// TIA Portal project "PLCSIM15-sort-height-basic_V17" (V17)
// Vorlageprojekt für das Buch mit Zielsystem S7-1200

(* hardware
DEVICE "S7-1200-Station_1"  S7-1200 Station
   slot 0: "Baugruppenträger_0"  Rack  V1.0
   slot 1: "PLC_1"  CPU 1211C DC/DC/DC  6ES7 211-1AE40-0XB0  V4.1
*)

// ===== PLC "PLC_1"  CPU 1211C DC/DC/DC =====

VAR_GLOBAL   // PLC tag table "Standard-Variablentabelle"
   "Tag_1" AT %A0.0 : Bool;
   "Tag_2" AT %E0.0 : Bool;
   "Tag_3" AT %E0.1 : Bool;
   "Warning Light" AT %Q1.2 : Bool;
END_VAR

VAR_GLOBAL   // PLC tag table "Tag table_1"
   "I_High_sensor" AT %I0.0 : Bool;
   "I_Low_sensor" AT %I0.1 : Bool;
   "I_Pallet_sensor" AT %I0.2 : Bool;
   "I_Loaded" AT %I0.3 : Bool;
   "I_At_left_entry" AT %I0.4 : Bool;
   "I_At_left_exit" AT %I0.5 : Bool;
   "I_At_right_entry" AT %I0.6 : Bool;
   "I_At_right_exit" AT %I0.7 : Bool;
   "O_Conveyor_entry" AT %Q0.0 : Bool;
   "O_Load" AT %Q0.1 : Bool;
   "O_Unload" AT %Q0.2 : Bool;
   "O_Transf_left" AT %Q0.3 : Bool;
   "O_Tranf_right" AT %Q0.4 : Bool;
   "O_Conveyor_left" AT %Q0.5 : Bool;
   "Loading" AT %M0.0 : Bool;
   "LoaderBusy" AT %M0.1 : Bool;
   "TransferingRight" AT %M0.2 : Bool;
   "TransferingLeft" AT %M0.3 : Bool;
   "HighBox" AT %M0.4 : Bool;
   "I_Start" AT %I1.0 : Bool;
   "I_Reset" AT %I1.1 : Bool;
   "I_Stop" AT %I1.2 : Bool;
   "I_Emergency" AT %I1.3 : Bool;
   "I_Auto" AT %I1.4 : Bool;
   "I_Factory_Running" AT %I1.5 : Bool;
   "O_Conveyor_right" AT %Q0.6 : Bool;
   "O_Start_light" AT %Q0.7 : Bool;
   "O_Reset_light" AT %Q1.0 : Bool;
   "O_Stop_light" AT %Q1.1 : Bool;
   "P_High_Sensor" AT %M1.0 : Bool;
   "P_Loading" AT %M1.1 : Bool;
   "P_At_left_entry" AT %M1.4 : Bool;
   "P_At_left_exit" AT %M1.5 : Bool;
   "P_At_right_entry" AT %M1.6 : Bool;
   "P_At_right_exit" AT %M1.7 : Bool;
   "P_Factory_Running" AT %M2.5 : Bool;
   "FactoryRestarting" AT %M0.5 : Bool;
END_VAR

// folder: System blocks/Program resources

DATA_BLOCK "RightCounter"   // DB1
{ S7_Optimized_Access := 'TRUE' }
AUTHOR : Simatic
FAMILY : IEC
NAME : CNTR
VERSION : 1.0
// stored: InstanceOfName IEC_COUNTER
"IEC_COUNTER"
BEGIN
END_DATA_BLOCK

DATA_BLOCK "LeftCounter"   // DB2
{ S7_Optimized_Access := 'TRUE' }
AUTHOR : Simatic
FAMILY : IEC
NAME : CNTR
VERSION : 1.0
// stored: InstanceOfName IEC_COUNTER
"IEC_COUNTER"
BEGIN
END_DATA_BLOCK

// folder: (top level)

FUNCTION "MHJ-PLC-Lab-Function-S71200" : Void   // FC9000, SCL
{ S7_Optimized_Access := 'TRUE' }
VERSION : 0.1
   VAR_TEMP
      rdTimeReturn : Int;
      outputTime : DTL;
      SyncVal : Byte;
      forVal : Int;
      forVal_2 : Int;
      Value : Byte;
   END_VAR
   VAR CONSTANT
      CompVal : Byte := 16#34;
      Value_01 : Byte := 16#11;
      Value_01_DW : DWord := 16#A165_D992;
      Value_02_DW : DWord := 16#58BE_4401;
   END_VAR
BEGIN

   #Value:=PEEK(area := 16#82,
        dbNumber := 0,
        byteOffset := 511);
   #Value := #Value + 1;

   POKE(area := 16#82,
        dbNumber := 0,
        byteOffset := 511,
        value := #Value);

   POKE(area:=16#81,
        dbNumber:=0,
        byteOffset:=1016,
        value:=#Value_01_DW);
   POKE(area := 16#81,
        dbNumber := 0,
        byteOffset := 1020,
        value := #Value_02_DW);

   POKE(area := 16#81,
        dbNumber := 0,
        byteOffset := 511,
        value := B#16#00);

   FOR #forVal := 0 TO 120 DO
       FOR #forVal_2:=0 TO 10 DO
           #rdTimeReturn:=RD_SYS_T(#outputTime);
           #rdTimeReturn := WR_SYS_T(#outputTime);
           #rdTimeReturn := RD_SYS_T(#outputTime);
           #rdTimeReturn := WR_SYS_T(#outputTime);
       END_FOR;
       #SyncVal:= PEEK(area := 16#81,
                      dbNumber := 0,
                      byteOffset := 511);
       IF #SyncVal = #CompVal THEN
          GOTO M_1;
       END_IF;
   END_FOR;
   RETURN;

   M_1:
   POKE(area := 16#81,
        dbNumber := 0,
        byteOffset := 511,
        value := B#16#0);
END_FUNCTION

ORGANIZATION_BLOCK "Main"   // OB1, LAD, ProgramCycle
TITLE = "Main Program Sweep (Cycle)"
{ S7_Optimized_Access := 'TRUE' }
VERSION : 0.1
   VAR_INPUT
      Initial_Call : Bool;   // Initial call of this OB
      Remanence : Bool;   // =True, if remanent data are available
   END_VAR
   VAR_TEMP   // added for the SCL form of the ladder/FBD networks
      _w1 : Bool;
   END_VAR
BEGIN

REGION Network 1: Connection block for PLCSIM communications. Don't delete this network!
   // Im Netzwerk 1 wird der Konnektierungsbaustein für PLC-Lab aufgerufen.
   // Dieser Aufruf darf nicht entfernt werden!
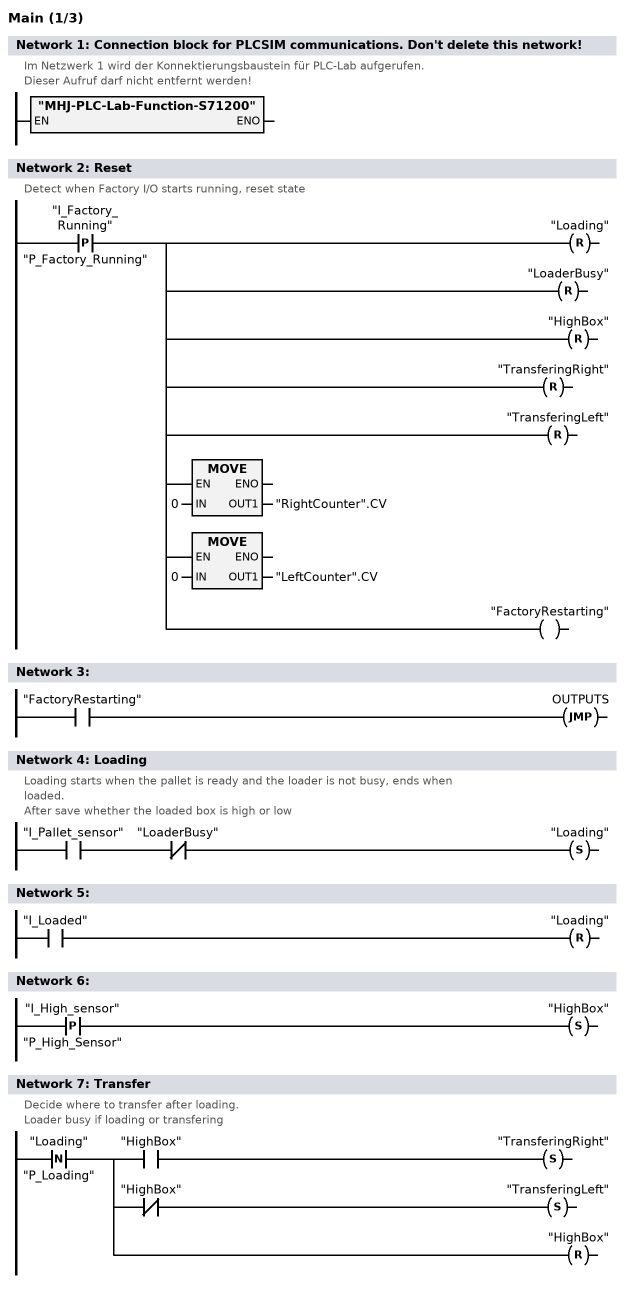
   RUNG wire#powerrail
      "MHJ-PLC-Lab-Function-S71200"()
   END_RUNG
   // the same network as SCL:
   "MHJ-PLC-Lab-Function-S71200"();
END_REGION

REGION Network 2: Reset
   // Detect when Factory I/O starts running, reset state
   RUNG wire#powerrail
      P_Contact(operand := "I_Factory_Running", bit := "P_Factory_Running")
      wire#w1
      R_Coil( "Loading" )
   END_RUNG
   RUNG wire#w1
      R_Coil( "LoaderBusy" )
   END_RUNG
   RUNG wire#w1
      R_Coil( "HighBox" )
   END_RUNG
   RUNG wire#w1
      R_Coil( "TransferingRight" )
   END_RUNG
   RUNG wire#w1
      R_Coil( "TransferingLeft" )
   END_RUNG
   RUNG wire#w1
      { S7_GenerateENO := "TRUE" } Move(in := 0, out1 => "RightCounter".CV)
   END_RUNG
   RUNG wire#w1
      { S7_GenerateENO := "TRUE" } Move(in := 0, out1 => "LeftCounter".CV)
   END_RUNG
   RUNG wire#w1
      Coil( "FactoryRestarting" )
   END_RUNG
   // the same network as SCL:
   #_w1 := "I_Factory_Running" AND NOT "P_Factory_Running";   // rising edge of "I_Factory_Running"
   "P_Factory_Running" := "I_Factory_Running";
   IF #_w1 THEN
       "Loading" := FALSE;
       "LoaderBusy" := FALSE;
       "HighBox" := FALSE;
       "TransferingRight" := FALSE;
       "TransferingLeft" := FALSE;
       "RightCounter".CV := 0;
       "LeftCounter".CV := 0;
   END_IF;
   "FactoryRestarting" := #_w1;
END_REGION

REGION Network 3
   RUNG wire#powerrail
      Contact( "FactoryRestarting" )
      JumpCoil( OUTPUTS )
   END_RUNG
   // the same network as SCL:
   IF "FactoryRestarting" THEN GOTO OUTPUTS; END_IF;
END_REGION

REGION Network 4: Loading
   // Loading starts when the pallet is ready and the loader is not busy, ends when 
   // loaded.
   // After save whether the loaded box is high or low
   RUNG wire#powerrail
      Contact( "I_Pallet_sensor" )
      I_Contact( "LoaderBusy" )
      S_Coil( "Loading" )
   END_RUNG
   // the same network as SCL:
   IF "I_Pallet_sensor" AND NOT "LoaderBusy" THEN "Loading" := TRUE; END_IF;
END_REGION

REGION Network 5
   RUNG wire#powerrail
      Contact( "I_Loaded" )
      R_Coil( "Loading" )
   END_RUNG
   // the same network as SCL:
   IF "I_Loaded" THEN "Loading" := FALSE; END_IF;
END_REGION

REGION Network 6
   RUNG wire#powerrail
      P_Contact(operand := "I_High_sensor", bit := "P_High_Sensor")
      S_Coil( "HighBox" )
   END_RUNG
   // the same network as SCL:
   #_w1 := "I_High_sensor" AND NOT "P_High_Sensor";   // rising edge of "I_High_sensor"
   "P_High_Sensor" := "I_High_sensor";
   IF #_w1 THEN "HighBox" := TRUE; END_IF;
END_REGION

REGION Network 7: Transfer
   // Decide where to transfer after loading.
   // Loader busy if loading or transfering
   RUNG wire#powerrail
      N_Contact(operand := "Loading", bit := "P_Loading")
      wire#w1
      Contact( "HighBox" )
      S_Coil( "TransferingRight" )
   END_RUNG
   RUNG wire#w1
      I_Contact( "HighBox" )
      S_Coil( "TransferingLeft" )
   END_RUNG
   RUNG wire#w1
      R_Coil( "HighBox" )
   END_RUNG
   // the same network as SCL:
   #_w1 := NOT "Loading" AND "P_Loading";   // falling edge of "Loading"
   "P_Loading" := "Loading";
   IF #_w1 AND "HighBox" THEN "TransferingRight" := TRUE; END_IF;
   IF #_w1 AND NOT "HighBox" THEN "TransferingLeft" := TRUE; END_IF;
   IF #_w1 THEN "HighBox" := FALSE; END_IF;
END_REGION

REGION Network 8
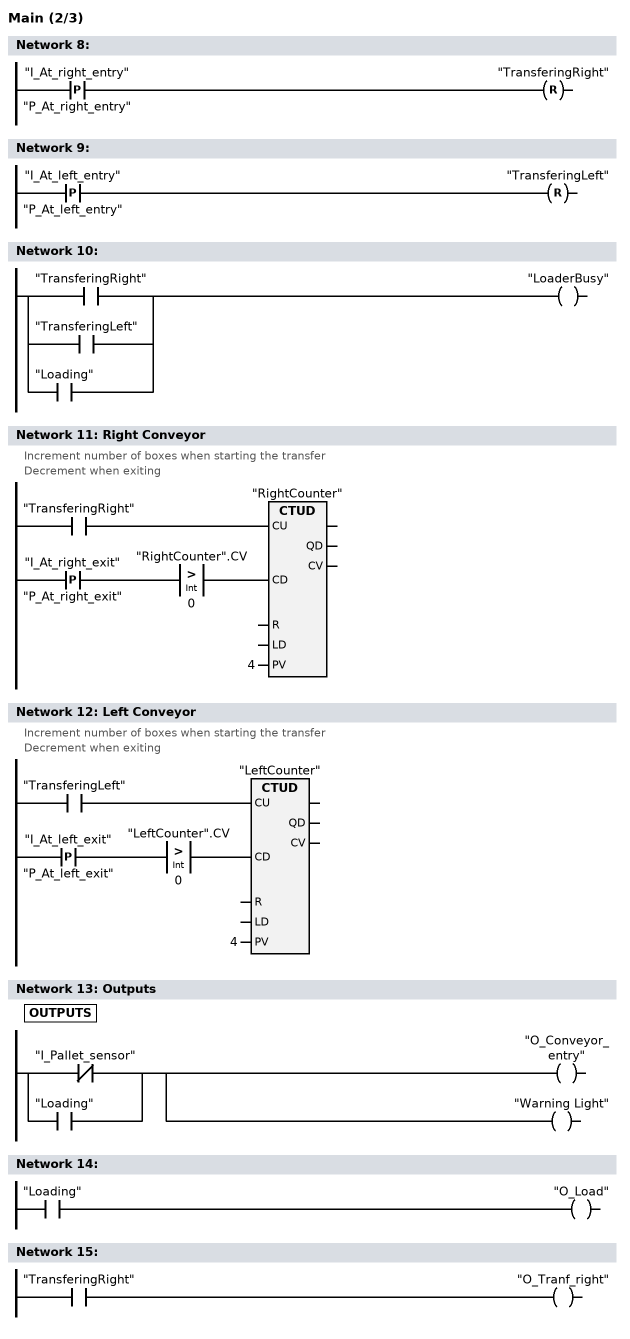
   RUNG wire#powerrail
      P_Contact(operand := "I_At_right_entry", bit := "P_At_right_entry")
      R_Coil( "TransferingRight" )
   END_RUNG
   // the same network as SCL:
   #_w1 := "I_At_right_entry" AND NOT "P_At_right_entry";   // rising edge of "I_At_right_entry"
   "P_At_right_entry" := "I_At_right_entry";
   IF #_w1 THEN "TransferingRight" := FALSE; END_IF;
END_REGION

REGION Network 9
   RUNG wire#powerrail
      P_Contact(operand := "I_At_left_entry", bit := "P_At_left_entry")
      R_Coil( "TransferingLeft" )
   END_RUNG
   // the same network as SCL:
   #_w1 := "I_At_left_entry" AND NOT "P_At_left_entry";   // rising edge of "I_At_left_entry"
   "P_At_left_entry" := "I_At_left_entry";
   IF #_w1 THEN "TransferingLeft" := FALSE; END_IF;
END_REGION

REGION Network 10
   RUNG wire#powerrail
      Contact( "TransferingRight" )
      wire#w1
      Coil( "LoaderBusy" )
   END_RUNG
   RUNG wire#powerrail
      Contact( "TransferingLeft" )
   END_RUNG wire#w1
   RUNG wire#powerrail
      Contact( "Loading" )
   END_RUNG wire#w1
   // the same network as SCL:
   "LoaderBusy" := "TransferingRight" OR "TransferingLeft" OR "Loading";
END_REGION

REGION Network 11: Right Conveyor
   // Increment number of boxes when starting the transfer
   // Decrement when exiting
   #_w1 := "I_At_right_exit" AND NOT "P_At_right_exit";   // rising edge of "I_At_right_exit"
   "P_At_right_exit" := "I_At_right_exit";
   "RightCounter".CTUD(CU := "TransferingRight", CD := #_w1 AND ("RightCounter".CV > 0), PV := 4);
END_REGION

REGION Network 12: Left Conveyor
   // Increment number of boxes when starting the transfer
   // Decrement when exiting
   #_w1 := "I_At_left_exit" AND NOT "P_At_left_exit";   // rising edge of "I_At_left_exit"
   "P_At_left_exit" := "I_At_left_exit";
   "LeftCounter".CTUD(CU := "TransferingLeft", CD := #_w1 AND ("LeftCounter".CV > 0), PV := 4);
END_REGION

REGION Network 13: Outputs
   Label( OUTPUTS )
   RUNG wire#powerrail
      I_Contact( "I_Pallet_sensor" )
      wire#w1
      Coil( "O_Conveyor_entry" )
   END_RUNG
   RUNG wire#powerrail
      Contact( "Loading" )
   END_RUNG wire#w1
   RUNG wire#w1
      Coil( "Warning Light" )
   END_RUNG
   // the same network as SCL:
   OUTPUTS:
   "O_Conveyor_entry" := NOT "I_Pallet_sensor" OR "Loading";
   "Warning Light" := "O_Conveyor_entry";
END_REGION

REGION Network 14
   RUNG wire#powerrail
      Contact( "Loading" )
      Coil( "O_Load" )
   END_RUNG
   // the same network as SCL:
   "O_Load" := "Loading";
END_REGION

REGION Network 15
   RUNG wire#powerrail
      Contact( "TransferingRight" )
      Coil( "O_Tranf_right" )
   END_RUNG
   // the same network as SCL:
   "O_Tranf_right" := "TransferingRight";
END_REGION

REGION Network 16
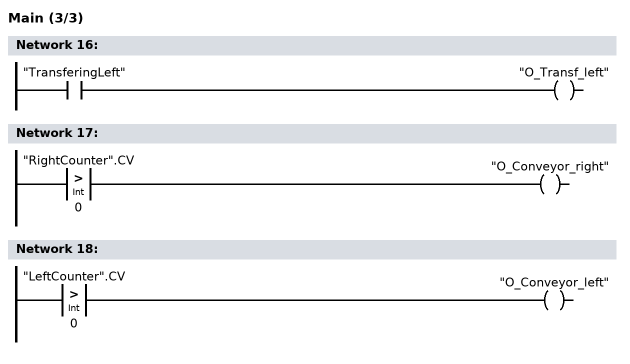
   RUNG wire#powerrail
      Contact( "TransferingLeft" )
      Coil( "O_Transf_left" )
   END_RUNG
   // the same network as SCL:
   "O_Transf_left" := "TransferingLeft";
END_REGION

REGION Network 17
   RUNG wire#powerrail
      { S7_Templates := "SrcType := Int" } GT_Contact(in1 := "RightCounter".CV, in2 := 0)
      Coil( "O_Conveyor_right" )
   END_RUNG
   // the same network as SCL:
   "O_Conveyor_right" := "RightCounter".CV > 0;
END_REGION

REGION Network 18
   RUNG wire#powerrail
      { S7_Templates := "SrcType := Int" } GT_Contact(in1 := "LeftCounter".CV, in2 := 0)
      Coil( "O_Conveyor_left" )
   END_RUNG
   // the same network as SCL:
   "O_Conveyor_left" := "LeftCounter".CV > 0;
END_REGION
END_ORGANIZATION_BLOCK